FUNCTION_BLOCK EffLoLoFlowMng (* CAT Function Block Type *)
  (* Standard: 61499-2 *)
  (* Version 0.0, 7/13/2026, Schneider Electric, template *)
  PACKAGE SE.Nereda;
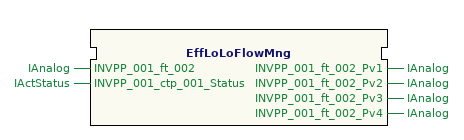
  SOCKETS
    INVPP_001_ft_002 : IAnalog;
    INVPP_001_ctp_001_Status : IActStatus;
  END_SOCKETS
  PLUGS
    INVPP_001_ft_002_Pv1 : IAnalog;
    INVPP_001_ft_002_Pv2 : IAnalog;
    INVPP_001_ft_002_Pv3 : IAnalog;
    INVPP_001_ft_002_Pv4 : IAnalog;
  END_PLUGS
  (* 01 - FUNCTIONNAL INPUT INTERFACE *)
  (* 05 - LOGIC *)
  (* 03 - FIELD INTERFACE *)
  (* 02 - FUNCTIONNAL OUTPUT INTERFACE *)
  FBS
    NVPP_001_ft_002_Status : decodeStatus;
    Pv1 : encodeStatus;
    D_Pv1 : DelayedActive(pin_4E076A4928A0DFEF := TRUE, pin_1CE054BDD0AD4DEB := T#1m);
    LoLoFlow : AND_550FE6D62F509EB3; {SET_ATTRIBUTE(Configuration.GenericFBType.InterfaceParams, Runtime.Standard#CNT:=3;OUT:BOOL)}
    Pv2 : encodeStatus;
    Pv3 : encodeStatus;
    Pv4 : encodeStatus;
    NotReady : NOT_42C76073DCEB1A7A; {SET_ATTRIBUTE(Configuration.GenericFBType.InterfaceParams, Runtime.Standard#CNT:=1;OUT${CNT$}:BOOL)}
  END_FBS
  EVENT_CONNECTIONS
    INVPP_001_ft_002.REQ_STATUS TO NVPP_001_ft_002_Status.REQ;
    Pv1.CNF TO INVPP_001_ft_002_Pv1.REQ_STATUS;
    INVPP_001_ctp_001_Status.14377629A1F197A9 TO D_Pv1.C451626F7187F42D;
    Pv2.CNF TO INVPP_001_ft_002_Pv2.REQ_STATUS;
    Pv3.CNF TO INVPP_001_ft_002_Pv3.REQ_STATUS;
    Pv4.CNF TO INVPP_001_ft_002_Pv4.REQ_STATUS;
    INVPP_001_ft_002.REQ TO INVPP_001_ft_002_Pv1.REQ;
    INVPP_001_ft_002.REQ TO INVPP_001_ft_002_Pv2.REQ;
    INVPP_001_ft_002.REQ TO INVPP_001_ft_002_Pv3.REQ;
    INVPP_001_ft_002.REQ TO INVPP_001_ft_002_Pv4.REQ;
    D_Pv1.DDA64CDC00519DA4 TO NotReady.REQ;
    NVPP_001_ft_002_Status.CNF TO NotReady.REQ;
    LoLoFlow.CNF TO Pv1.REQ;
    LoLoFlow.CNF TO Pv2.REQ;
    LoLoFlow.CNF TO Pv3.REQ;
    LoLoFlow.CNF TO Pv4.REQ;
    NotReady.CNF TO LoLoFlow.REQ;
  END_CONNECTIONS
  DATA_CONNECTIONS
    INVPP_001_ft_002.Status TO NVPP_001_ft_002_Status.Status;
    Pv1.Status TO INVPP_001_ft_002_Pv1.Status;
    INVPP_001_ctp_001_Status.D41A46B14EF7208D TO D_Pv1.19546B227DE05AED;
    INVPP_001_ctp_001_Status.D41A46B14EF7208D TO D_Pv1.45767490F5BA3A44;
    Pv2.Status TO INVPP_001_ft_002_Pv2.Status;
    Pv3.Status TO INVPP_001_ft_002_Pv3.Status;
    Pv4.Status TO INVPP_001_ft_002_Pv4.Status;
    NVPP_001_ft_002_Status.StateAlarm TO Pv1.StateAlarm;
    NVPP_001_ft_002_Status.HiHiAlarm TO Pv1.HiHiAlarm;
    NVPP_001_ft_002_Status.HiAlarm TO Pv1.HiAlarm;
    NVPP_001_ft_002_Status.LoAlarm TO Pv1.LoAlarm;
    NVPP_001_ft_002_Status.DevAlarm TO Pv1.DevAlarm;
    NVPP_001_ft_002_Status.DevHi TO Pv1.DevHi;
    NVPP_001_ft_002_Status.DevLo TO Pv1.DevLo;
    NVPP_001_ft_002_Status.RocAlarm TO Pv1.RocAlarm;
    NVPP_001_ft_002_Status.RocHi TO Pv1.RocHi;
    NVPP_001_ft_002_Status.RocLo TO Pv1.RocLo;
    NVPP_001_ft_002_Status.MinActive TO Pv1.MinActive;
    NVPP_001_ft_002_Status.MaxActive TO Pv1.MaxActive;
    NVPP_001_ft_002_Status.FailAlarm TO Pv1.FailAlarm;
    NVPP_001_ft_002_Status.CurrentNotOkAlarm TO Pv1.CurrentNotOkAlarm;
    NVPP_001_ft_002_Status.VoltageNotOkAlarm TO Pv1.VoltageNotOkAlarm;
    NVPP_001_ft_002_Status.LoBatteryAlarm TO Pv1.LoBatteryAlarm;
    NVPP_001_ft_002_Status.LoGasAlarm TO Pv1.LoGasAlarm;
    NVPP_001_ft_002_Status.TempHiAlarm TO Pv1.TempHiAlarm;
    NVPP_001_ft_002_Status.PressHiAlarm TO Pv1.PressHiAlarm;
    NVPP_001_ft_002_Status.StateAlarm TO Pv2.StateAlarm;
    NVPP_001_ft_002_Status.HiHiAlarm TO Pv2.HiHiAlarm;
    NVPP_001_ft_002_Status.HiAlarm TO Pv2.HiAlarm;
    NVPP_001_ft_002_Status.LoAlarm TO Pv2.LoAlarm;
    NVPP_001_ft_002_Status.DevAlarm TO Pv2.DevAlarm;
    NVPP_001_ft_002_Status.DevHi TO Pv2.DevHi;
    NVPP_001_ft_002_Status.DevLo TO Pv2.DevLo;
    NVPP_001_ft_002_Status.RocAlarm TO Pv2.RocAlarm;
    NVPP_001_ft_002_Status.RocHi TO Pv2.RocHi;
    NVPP_001_ft_002_Status.RocLo TO Pv2.RocLo;
    NVPP_001_ft_002_Status.MinActive TO Pv2.MinActive;
    NVPP_001_ft_002_Status.MaxActive TO Pv2.MaxActive;
    NVPP_001_ft_002_Status.FailAlarm TO Pv2.FailAlarm;
    NVPP_001_ft_002_Status.CurrentNotOkAlarm TO Pv2.CurrentNotOkAlarm;
    NVPP_001_ft_002_Status.VoltageNotOkAlarm TO Pv2.VoltageNotOkAlarm;
    NVPP_001_ft_002_Status.LoBatteryAlarm TO Pv2.LoBatteryAlarm;
    NVPP_001_ft_002_Status.LoGasAlarm TO Pv2.LoGasAlarm;
    NVPP_001_ft_002_Status.TempHiAlarm TO Pv2.TempHiAlarm;
    NVPP_001_ft_002_Status.PressHiAlarm TO Pv2.PressHiAlarm;
    NVPP_001_ft_002_Status.StateAlarm TO Pv3.StateAlarm;
    NVPP_001_ft_002_Status.HiHiAlarm TO Pv3.HiHiAlarm;
    NVPP_001_ft_002_Status.HiAlarm TO Pv3.HiAlarm;
    NVPP_001_ft_002_Status.LoAlarm TO Pv3.LoAlarm;
    NVPP_001_ft_002_Status.DevAlarm TO Pv3.DevAlarm;
    NVPP_001_ft_002_Status.DevHi TO Pv3.DevHi;
    NVPP_001_ft_002_Status.DevLo TO Pv3.DevLo;
    NVPP_001_ft_002_Status.RocAlarm TO Pv3.RocAlarm;
    NVPP_001_ft_002_Status.RocHi TO Pv3.RocHi;
    NVPP_001_ft_002_Status.RocLo TO Pv3.RocLo;
    NVPP_001_ft_002_Status.MinActive TO Pv3.MinActive;
    NVPP_001_ft_002_Status.MaxActive TO Pv3.MaxActive;
    NVPP_001_ft_002_Status.FailAlarm TO Pv3.FailAlarm;
    NVPP_001_ft_002_Status.CurrentNotOkAlarm TO Pv3.CurrentNotOkAlarm;
    NVPP_001_ft_002_Status.VoltageNotOkAlarm TO Pv3.VoltageNotOkAlarm;
    NVPP_001_ft_002_Status.LoBatteryAlarm TO Pv3.LoBatteryAlarm;
    NVPP_001_ft_002_Status.LoGasAlarm TO Pv3.LoGasAlarm;
    NVPP_001_ft_002_Status.TempHiAlarm TO Pv3.TempHiAlarm;
    NVPP_001_ft_002_Status.PressHiAlarm TO Pv3.PressHiAlarm;
    NVPP_001_ft_002_Status.StateAlarm TO Pv4.StateAlarm;
    NVPP_001_ft_002_Status.HiHiAlarm TO Pv4.HiHiAlarm;
    NVPP_001_ft_002_Status.HiAlarm TO Pv4.HiAlarm;
    NVPP_001_ft_002_Status.LoAlarm TO Pv4.LoAlarm;
    NVPP_001_ft_002_Status.DevAlarm TO Pv4.DevAlarm;
    NVPP_001_ft_002_Status.DevHi TO Pv4.DevHi;
    NVPP_001_ft_002_Status.DevLo TO Pv4.DevLo;
    NVPP_001_ft_002_Status.RocAlarm TO Pv4.RocAlarm;
    NVPP_001_ft_002_Status.RocHi TO Pv4.RocHi;
    NVPP_001_ft_002_Status.RocLo TO Pv4.RocLo;
    NVPP_001_ft_002_Status.MinActive TO Pv4.MinActive;
    NVPP_001_ft_002_Status.MaxActive TO Pv4.MaxActive;
    NVPP_001_ft_002_Status.FailAlarm TO Pv4.FailAlarm;
    NVPP_001_ft_002_Status.CurrentNotOkAlarm TO Pv4.CurrentNotOkAlarm;
    NVPP_001_ft_002_Status.VoltageNotOkAlarm TO Pv4.VoltageNotOkAlarm;
    NVPP_001_ft_002_Status.LoBatteryAlarm TO Pv4.LoBatteryAlarm;
    NVPP_001_ft_002_Status.LoGasAlarm TO Pv4.LoGasAlarm;
    NVPP_001_ft_002_Status.TempHiAlarm TO Pv4.TempHiAlarm;
    NVPP_001_ft_002_Status.PressHiAlarm TO Pv4.PressHiAlarm;
    INVPP_001_ft_002.Value TO INVPP_001_ft_002_Pv1.Value;
    INVPP_001_ft_002.ValueMin TO INVPP_001_ft_002_Pv1.ValueMin;
    INVPP_001_ft_002.ValueMax TO INVPP_001_ft_002_Pv1.ValueMax;
    INVPP_001_ft_002.Value TO INVPP_001_ft_002_Pv2.Value;
    INVPP_001_ft_002.ValueMin TO INVPP_001_ft_002_Pv2.ValueMin;
    INVPP_001_ft_002.ValueMax TO INVPP_001_ft_002_Pv2.ValueMax;
    INVPP_001_ft_002.Value TO INVPP_001_ft_002_Pv3.Value;
    INVPP_001_ft_002.ValueMin TO INVPP_001_ft_002_Pv3.ValueMin;
    INVPP_001_ft_002.ValueMax TO INVPP_001_ft_002_Pv3.ValueMax;
    INVPP_001_ft_002.Value TO INVPP_001_ft_002_Pv4.Value;
    INVPP_001_ft_002.ValueMin TO INVPP_001_ft_002_Pv4.ValueMin;
    INVPP_001_ft_002.ValueMax TO INVPP_001_ft_002_Pv4.ValueMax;
    D_Pv1.614F3125208254F6 TO LoLoFlow.IN1;
    NVPP_001_ft_002_Status.LoLoAlarm TO LoLoFlow.IN2;
    LoLoFlow.OUT TO Pv1.LoLoAlarm;
    LoLoFlow.OUT TO Pv2.LoLoAlarm;
    LoLoFlow.OUT TO Pv3.LoLoAlarm;
    LoLoFlow.OUT TO Pv4.LoLoAlarm;
    NotReady.OUT1 TO LoLoFlow.IN3;
    INVPP_001_ctp_001_Status.9E0B44559326BEAF TO NotReady.IN1;
  END_CONNECTIONS
END_FUNCTION_BLOCK
